// TIA Portal V15.1 export
// export: Created 2019-03-26T09:50:17.9382414Z, ExportSetting WithDefaults, DisplayName Totally Integrated Automation Portal, DisplayVersion V15.1, DisplayName TIA Portal Openness, DisplayVersion V15.1, DisplayName STEP 7 Professional, DisplayVersion V15.1, DisplayName WinCC Advanced, DisplayVersion V15.1
Screen "Bild_1"  800x480, Number=2
  ScreenLayer 
    TextField "Textfeld_1" at 74,206 size 658x66  Text="Hello from TIA Openness!"
